TYPE ST_HW_OutputsLowLiftUnit :
(**************************************************************************************
 * 	Application		:	BoxControl Framework
 *	Revision		:	$Revision: 417092 $
 *	Revision date	:	$Date: 2018-11-14 12:58:58 +0100 (Mi., 14 Nov 2018) $
 *	Last changed by	:	$Author: q8aberh $
 *	URL				:	$URL: http://almscdc.swisslog.com/repo/SWPD/Development/ProMove/02_Controls/ProBox/03_Implementation/01_DevelopmentProject/01_Software/ProBox_COE/ProBox_DevProj_v1.0/PLC_1/20_Product/10_App/12_E_Functions/11_ProBox/21_LowLiftUnit/10_App/01_DUTs/ST_HW_Ou $
 *
 *	Purpose			:	HW outputs of the dummy function
 *
 * ------------------------------------------------------------------------------------
 *	Copyright Swisslog [IP AG], Switzerland. All rights reserved.
 * 
 * ------------------------------------------------------------------------------------
 *	
 * 	Revision History: 
 *
 * 	VERSION			DATE			INITIALS			DESCRIPTION
 *	0.1				01.01.2001		swl					Example
 *
 **************************************************************************************)	
STRUCT
	Drive_Run_Up			: BOOL; // Drive run command lift up
	Drive_Run_Down			: BOOL; // Drive run command lift down
	Drive_Low_UpDown		: BOOL; // Drive low speed command lift
	Drive_Creep_UpDown		: BOOL; // Drive creep speed command lift	
	Lamp_ResetLightgrid		: BOOL; // Lamp reset lightgrid
END_STRUCT
END_TYPE

(* stored: Version 1.1.0.1, ProductVersion 3.1.4020.6
   DUT ST_HW_OutputsLowLiftUnit: Id {d07258dc-e92d-43dd-851e-82bc43332a0b} *)
